// TIA Portal project "lab_02" (V16)

(* hardware
DEVICE "S71500/ET200MP station_1"  S7-1500 station
   slot 0: "Perfil soporte_0"  Rack  6ES7 590-1***0-0AA0
   slot 1: "PLC_1"  CPU 1515-2 PN  6ES7 515-2AM02-0AB0  V2.8
      slot 3: "Display de la CPU_1"  6ES7591-1BA00-0AA0
      slot 32768: "Interfaz PROFINET_1"  X1
         slot 32769: "Puerto_1"  X1 P1
         slot 32770: "Puerto_2"  X1 P2
      slot 33024: "Interfaz PROFINET_2"  X2
         slot 33025: "Puerto_1"  X2 P1
      slot 34817: "Virtual CP interface port_1"  Virtual CP interface port  Virtual CP interface port
*)

// ===== PLC "PLC_1"  CPU 1515-2 PN =====

VAR_GLOBAL   // PLC tag table "Tabla de variables estándar"
   "System_Byte" AT %MB1 : Byte;
   "FirstScan" AT %M1.0 : Bool;
   "DiagStatusUpdate" AT %M1.1 : Bool;
   "AlwaysTRUE" AT %M1.2 : Bool;
   "AlwaysFALSE" AT %M1.3 : Bool;
   "Clock_Byte" AT %MB0 : Byte;
   "Clock_10Hz" AT %M0.0 : Bool;
   "Clock_5Hz" AT %M0.1 : Bool;
   "Clock_2.5Hz" AT %M0.2 : Bool;
   "Clock_2Hz" AT %M0.3 : Bool;
   "Clock_1.25Hz" AT %M0.4 : Bool;
   "Clock_1Hz" AT %M0.5 : Bool;
   "Clock_0.625Hz" AT %M0.6 : Bool;
   "Clock_0.5Hz" AT %M0.7 : Bool;
   "Input0_0" AT %I0.0 : Bool;
   "Tag_2" AT %M2.0 : Bool;
   "Marca2_1" AT %M2.1 : Bool;
END_VAR

DATA_BLOCK "Logo_S7"   // DB1
{ S7_Optimized_Access := 'FALSE' }
VERSION : 0.1
   VAR
      i1 : Bool;
      i2 : Bool;
      i3 : Bool;
      i4 : Bool;
      i5 : Bool;
      i6 : Bool;
      i7 : Bool;
      i8 : Bool;
      Q1 : Bool;
      Q2 : Bool;
      Q3 : Bool;
      Q4 : Bool;
      VW2 : Int;
      VW4 : Int;
   END_VAR
BEGIN
END_DATA_BLOCK

FUNCTION "FC_Logo_S7" : Void   // FC1, FBD
{ S7_Optimized_Access := 'TRUE' }
VERSION : 0.1
   VAR_TEMP   // added for the SCL form of the ladder/FBD networks
      _w1 : Bool;
   END_VAR
BEGIN

REGION Network 1: Activar salida Q1 del logo 8 desde la entrada i0.0 o la marca 2.0 del PLC 1200
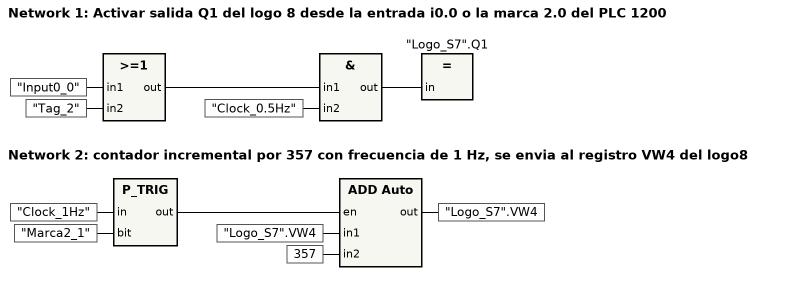
   "Logo_S7".Q1 := ("Input0_0" OR "Tag_2") AND "Clock_0.5Hz";
END_REGION

REGION Network 2: contador incremental por 357 con frecuencia de 1 Hz, se envia al registro VW4 del logo8
   #_w1 := "Clock_1Hz" AND NOT "Marca2_1";   // rising edge
   "Marca2_1" := "Clock_1Hz";
   IF #_w1 THEN "Logo_S7".VW4 := "Logo_S7".VW4 + 357; END_IF;
END_REGION
END_FUNCTION

ORGANIZATION_BLOCK "Main"   // OB1, LAD, ProgramCycle
TITLE = "Main Program Sweep (Cycle)"
{ S7_Optimized_Access := 'TRUE' }
VERSION : 0.1
   VAR_INPUT
      Initial_Call : Bool;   // Initial call of this OB
      Remanence : Bool;   // =True, if remanent data are available
   END_VAR
BEGIN

REGION Network 1
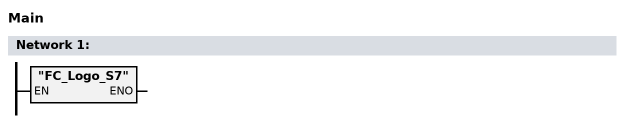
   RUNG wire#powerrail
      "FC_Logo_S7"()
   END_RUNG
   // the same network as SCL:
   "FC_Logo_S7"();
END_REGION
END_ORGANIZATION_BLOCK